// TIA Portal V20 export
TYPE "UDT_Service_Value"
   STRUCT
      Analog : Real;   // Analog value
      Digital : DInt;   // Digital value
      Binary : Bool;   // Binary value
      "String" : String[40];   // String value
   END_STRUCT;
END_TYPE
